# B&R Automation Studio project CarWash
Automation Studio 

## Configuration Config1

### Task classes (Cpu.sw)
```
Cyclic#1 (cycle 10000 us, tolerance 10000 us):
  Auxillary <- Source.Auxillary.Auxillary.prg
  MainCtrl <- Source.MainCtrl.MainCtrl.prg
  HPolish <- Source.Hpol.HPolish.prg
  EntryCtrl <- Source.Entrance.EntryCtrl.prg
  ChemCtrl <- Source.Chemicals.ChemCtrl.prg
  HPWater <- Source.HPWater.HPWater.prg
  HBrushCtrl <- Source.HBrush.HBrushCtrl.prg
  VBrushCtrl <- Source.VBrush.VBrushCtrl.prg
  UBCtrl <- Source.OptUnderBody.UBCtrl.prg
  VPolishCtr <- Source.OptVpolish.VPolishCtrl.prg
  WaxCtrl <- Source.OptWax.WaxCtrl.prg
  DryHCtrl <- Source.Drying.DryHCtrl.prg
  CarExit <- Source.CarExit.CarExit.prg
  AlarmCtrl <- Source.Infrastructure.AlarmCtrl.AlarmCtrl.prg
  DataCtrl <- Source.Infrastructure.DataCtrl.DataCtrl.prg
  RecipeCtrl <- Source.Infrastructure.RecipeCtrl.RecipeCtrl.prg
  VisuCtrl <- Source.VisuCtrl.VisuCtrl.prg
Cyclic#4 (cycle 100000 us, tolerance 100000 us):
  ComTCP_P <- Libraries.ComTCP.ComTCP_P.prg
Libraries: ComTCP_L, AsTCP, operator, runtime, astime, standard, ArEventLog, AsBrStr
```

### Hardware
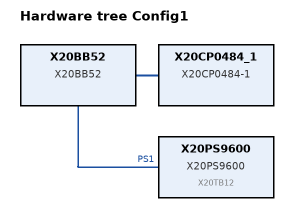
```
X20BB52 : X20BB52 v1.2.0.0
X20CP0484_1 : X20CP0484-1 v1.4.0.0  [SL -> X20BB52.SL1]
  Connector IF2:
    ActivateDevice = 1
  ConfigurationID = CarWashSimu_Config1
  Simulation = 1
  TimerDeviceType = SWIOTIMER
  Cyclic1Duration = 10000
  Cyclic1Tolerance = 10000
  Cyclic2Duration = 20000
  Cyclic2Tolerance = 20000
  Cyclic3Duration = 50000
  Cyclic3Tolerance = 50000
  Cyclic4Duration = 100000
  Cyclic4Tolerance = 100000
  Cyclic5Duration = 200000
  Cyclic5Tolerance = 200000
  Cyclic6Duration = 500000
  Cyclic6Tolerance = 500000
  Cyclic7Duration = 1000000
  Cyclic7Tolerance = 1000000
  Cyclic8Duration = 10000
  Cyclic8Tolerance = 30000000
  FileDevice1
  FileDeviceName1 = USER
  FileDevicePath1 = USER_PATH
X20PS9600 : X20PS9600 v1.6.0.0  [PS -> X20BB52.PS1; SS1 -> X20TB12.SS]
X20TB12 : X20TB12 v1.0.0.0
```

### PvMap.vvm - X20CP0484_1/PvMap.vvm
```iecst
VAR_CONFIG
<<<<<<< HEAD
	::CarExit:iExit.IO.doOrangeLight AT %Q.::ComTCP_SimOutputs.doExitOrangeLight; (*Insert your comment here...*)
	::CarExit:iExit.IO.doRedLight AT %Q.::ComTCP_SimOutputs.doExitRedLight; (*Insert your comment here...*)
	::ComTCP_SimOutputs.doExitGreenLight AT %Q.::ComTCP_SimOutputs.doExitGreenLight; (*Insert your comment here...*)
	::ComTCP_SimOutputs.doExitLiftDoorRelay AT %Q.::CarExit:iExit.IO.doRelayLiftDoor; (*Insert your comment here...*)
	::CarExit:iExit.IO.doRelayLowerdDoor AT %Q.::ComTCP_SimOutputs.doExitLowerDoorRelay; (*Insert your comment here...*)
	::MainCtrl:ScalDirt.y AT %Q.::ChemCtrl:iChem.IO.aoChemChemValve; (*Insert your comment here...*)
=======
	::VBrushCtrl:iVBrush.Par.LeftVel AT %Q.::ComTCP_SimOutputs.aoVBrushLVel; (*Insert your comment here...*)
	::VBrushCtrl:iVBrush.Par.RightVel AT %Q.::ComTCP_SimOutputs.aoVBrushRVel; (*Insert your comment here...*)
	::Auxillary:iAuxillary.doRelayConv AT %Q.::ComTCP_SimOutputs.doConvRelay; (*Insert your comment here...*)
	::ChemCtrl:iChem.IO.doChemWaterValve AT %Q.::ComTCP_SimOutputs.doChemWaterValve; (*Insert your comment here...*)
>>>>>>> edcf355ccd2dc5a058ed4214cc82538d90d7c920
	::ComTCP_SimInputs.aiEntranceSoilLevel AT %Q.::EntryCtrl:iEntry.IO.diSensSoilLvl; (*Insert your comment here...*)
	::ComTCP_SimInputs.aiVBrushLForceF AT %Q.::VBrushCtrl:iVBrush.IO.aiVBLForceF; (*Insert your comment here...*)
	::ComTCP_SimInputs.aiVBrushLForceS AT %Q.::VBrushCtrl:iVBrush.IO.aiVBLForceS; (*Insert your comment here...*)
	::ComTCP_SimInputs.aiVBrushRForceF AT %Q.::VBrushCtrl:iVBrush.IO.aiVBRForceF; (*Insert your comment here...*)
	::ComTCP_SimInputs.aiVBrushRForceS AT %Q.::VBrushCtrl:iVBrush.IO.aiVBRForceS; (*Insert your comment here...*)
	::ComTCP_SimInputs.diEmergencyStop AT %Q.::MainCtrl:gMain.Cmd.EStop; (*Insert your comment here...*)
	::ComTCP_SimInputs.diEntranceSensor AT %Q.::EntryCtrl:iEntry.IO.diSensEntry; (*Insert your comment here...*)
	::ComTCP_SimInputs.diHBrushSensor1 AT %Q.::HBrushCtrl:iHBrush.IO.diSensHB1; (*Insert your comment here...*)
	::ComTCP_SimInputs.diHBrushSensor2 AT %Q.::HBrushCtrl:iHBrush.IO.diSensHB2; (*Insert your comment here...*)
	::ComTCP_SimInputs.diHBrushSensor3 AT %Q.::HBrushCtrl:iHBrush.IO.diSensHB3; (*Insert your comment here...*)
	::ComTCP_SimInputs.diHBrushSensor4 AT %Q.::HBrushCtrl:iHBrush.IO.diSensHB4; (*Insert your comment here...*)
	::ComTCP_SimInputs.diHighPressSensor1 AT %Q.::HPWater:iHighPress.IO.diSensHP1; (*Insert your comment here...*)
	::ComTCP_SimInputs.diHighPressSensor2 AT %Q.::HPWater:iHighPress.IO.diSensHP2; (*Insert your comment here...*)
	::ComTCP_SimInputs.diHighPressSensor3 AT %Q.::HPWater:iHighPress.IO.diSensHP3; (*Insert your comment here...*)
	::ComTCP_SimInputs.diHighPressSensor4 AT %Q.::HPWater:iHighPress.IO.diSensHP4; (*Insert your comment here...*)
	::ComTCP_SimInputs.diHPolishSensor1 AT %Q.::HPolish:iHPolish.IO.diSensHPolish1; (*Insert your comment here...*)
	::ComTCP_SimInputs.diHPolishSensor2 AT %Q.::HPolish:iHPolish.IO.diSensHPolish2; (*Insert your comment here...*)
	::ComTCP_SimInputs.diHPolishSensor3 AT %Q.::HPolish:iHPolish.IO.diSensHPolish3; (*Insert your comment here...*)
	::ComTCP_SimInputs.diHPolishSensor4 AT %Q.::HPolish:iHPolish.IO.diSensHPolish4; (*Insert your comment here...*)
	::HBrushCtrl:iHBrush.IO.doRelayHBBrush AT %Q.::ComTCP_SimOutputs.doHBrushBrushRelay; (*Insert your comment here...*)
	::HBrushCtrl:iHBrush.IO.doRelayHBLift AT %Q.::ComTCP_SimOutputs.doHBrushLiftRelay; (*Insert your comment here...*)
	::HBrushCtrl:iHBrush.IO.doRelayHBLower AT %Q.::ComTCP_SimOutputs.doHBrushLowerRelay; (*Insert your comment here...*)
	::HBrushCtrl:iHBrush.IO.doValveHB AT %Q.::ComTCP_SimOutputs.doHBrushValve; (*Insert your comment here...*)
	::HPolish:iHPolish.IO.doRelayBrush AT %Q.::ComTCP_SimOutputs.doHPolishBrushRelay; (*Insert your comment here...*)
	::HPolish:iHPolish.IO.doRelayLift AT %Q.::ComTCP_SimOutputs.doHPolishLiftRelay; (*Insert your comment here...*)
	::HPolish:iHPolish.IO.doRelayLower AT %Q.::ComTCP_SimOutputs.doHPolishLowerRelay; (*Insert your comment here...*)
	::HPWater:iHighPress.IO.doRelayHPLift AT %Q.::ComTCP_SimOutputs.doHighPressLiftRelay; (*Insert your comment here...*)
	::HPWater:iHighPress.IO.doRelayHPLow AT %Q.::ComTCP_SimOutputs.doHighPressLowerRelay; (*Insert your comment here...*)
	::HPWater:iHighPress.IO.doRelayHPPump AT %Q.::ComTCP_SimOutputs.doHighPressPumpRelay; (*Insert your comment here...*)
	::HPWater:iHighPress.IO.doValveHP AT %Q.::ComTCP_SimOutputs.doHighPressValve; (*Insert your comment here...*)
	::MainCtrl:ScalDirt.y AT %Q.::ChemCtrl:iChem.IO.aoChemChemValve; (*Insert your comment here...*)
	::UBCtrl:iUBody.IO.doRelayPump AT %Q.::ComTCP_SimOutputs.doUnderbodyPumpRelay; (*Insert your comment here...*)
	::UBCtrl:iUBody.IO.doValveUB AT %Q.::ComTCP_SimOutputs.doUnderbodyValve; (*Insert your comment here...*)
	::VBrushCtrl:iVBrush.IO.doRelayVBLClose AT %Q.::ComTCP_SimOutputs.doVBrushRelayLClose; (*Insert your comment here...*)
	::VBrushCtrl:iVBrush.IO.doRelayVBLOpen AT %Q.::ComTCP_SimOutputs.doVBrushRelayLOpen; (*Insert your comment here...*)
	::VBrushCtrl:iVBrush.IO.doRelayVBRClose AT %Q.::ComTCP_SimOutputs.doVBrushRelayRClose; (*Insert your comment here...*)
	::VBrushCtrl:iVBrush.IO.doRelayVBROpen AT %Q.::ComTCP_SimOutputs.doVBrushRelayROpen; (*Insert your comment here...*)
<<<<<<< HEAD
	::VBrushCtrl:iVBrush.IO.doRelayVBLOpen AT %Q.::ComTCP_SimOutputs.doVBrushRelayLOpen; (*Insert your comment here...*)
	::ComTCP_SimInputs.aiVBrushLForceF AT %Q.::VBrushCtrl:iVBrush.IO.aiVBLForceF; (*Insert your comment here...*)
	::ComTCP_SimInputs.aiVBrushRForceF AT %Q.::VBrushCtrl:iVBrush.IO.aiVBRForceF; (*Insert your comment here...*)
	::ComTCP_SimInputs.aiVBrushLForceS AT %Q.::VBrushCtrl:iVBrush.IO.aiVBLForceS; (*Insert your comment here...*)
	::ComTCP_SimInputs.aiVBrushRForceS AT %Q.::VBrushCtrl:iVBrush.IO.aiVBRForceS; (*Insert your comment here...*)
	::ComTCP_SimInputs.diHDry1Sensor1 AT %Q.::DryHCtrl:iDry.IO.diSens1Dry1; (*Insert your comment here...*)
	::ComTCP_SimInputs.diHDry1Sensor2 AT %Q.::DryHCtrl:iDry.IO.diSens1Dry2; (*Insert your comment here...*)
	::ComTCP_SimInputs.diHDry1Sensor3 AT %Q.::DryHCtrl:iDry.IO.diSens1Dry3; (*Insert your comment here...*)
	::ComTCP_SimInputs.diHDry1Sensor4 AT %Q.::DryHCtrl:iDry.IO.diSens1Dry4; (*Insert your comment here...*)
	::ComTCP_SimInputs.diHDry2Sensor1 AT %Q.::DryHCtrl:iDry.IO.diSens2Dry1; (*Insert your comment here...*)
	::ComTCP_SimInputs.diHDry2Sensor2 AT %Q.::DryHCtrl:iDry.IO.diSens2Dry2; (*Insert your comment here...*)
	::ComTCP_SimInputs.diHDry2Sensor3 AT %Q.::DryHCtrl:iDry.IO.diSens2Dry3; (*Insert your comment here...*)
	::ComTCP_SimInputs.diHDry2Sensor4 AT %Q.::DryHCtrl:iDry.IO.diSens2Dry4; (*Insert your comment here...*)
	::DryHCtrl:iDry.IO.doRelayHD1Vent AT %Q.::ComTCP_SimOutputs.doHDry1VentRelay; (*Insert your comment here...*)
	::DryHCtrl:iDry.IO.doRelayHD1Heater AT %Q.::ComTCP_SimOutputs.doHDry1HeaterRelay; (*Insert your comment here...*)
	::DryHCtrl:iDry.IO.doRelayHD1Lower AT %Q.::ComTCP_SimOutputs.doHDry1LowerRelay; (*Insert your comment here...*)
	::DryHCtrl:iDry.IO.doRelayHD1Lift AT %Q.::ComTCP_SimOutputs.doHDry1LiftRelay; (*Insert your comment here...*)
	::DryHCtrl:iDry.IO.doRelayHD2Vent AT %Q.::ComTCP_SimOutputs.doHDry2VentRelay; (*Insert your comment here...*)
	::DryHCtrl:iDry.IO.doRelayHD2Heater AT %Q.::ComTCP_SimOutputs.doHDry2HeaterRelay; (*Insert your comment here...*)
	::DryHCtrl:iDry.IO.doRelayHD2Lower AT %Q.::ComTCP_SimOutputs.doHDry2LowerRelay; (*Insert your comment here...*)
	::DryHCtrl:iDry.IO.doRelayVDHeater AT %Q.::ComTCP_SimOutputs.doVDry1HeaterRelay; (*Insert your comment here...*)
	::DryHCtrl:iDry.IO.doRelayVDVent AT %Q.::ComTCP_SimOutputs.doVDry1VentRelay; (*Insert your comment here...*)
	::DryHCtrl:iDry.IO.doRelayHD2Lift AT %Q.::ComTCP_SimOutputs.doHDry2LiftRelay; (*Insert your comment here...*)
=======
	::WaxCtrl:iWax.IO.doValveWax AT %Q.::ComTCP_SimOutputs.doWaxValve; (*Insert your comment here...*)
	::WaxCtrl:iWax.IO.doRefillWax AT %Q.::ComTCP_SimOutputs.doWaxRefill; (*Insert your comment here...*)
	::WaxCtrl:iWax.IO.doRealyWaxPump AT %Q.::ComTCP_SimOutputs.doWaxPumpRelay; (*Insert your comment here...*)
>>>>>>> edcf355ccd2dc5a058ed4214cc82538d90d7c920
END_VAR
```

## Logical view

Binary libraries used (declarations not repeated): operator, runtime, astime, AsIecCon, AsTCP, standard, ArEventLog, AsBrStr, LoopConR, sys_lib, brsystem

### Package Logical/Libraries - Global libraries

### Library Logical/Libraries/ComTCP/ComTCP_L (ANSIC)
Depends on: AsTCP, operator, runtime, astime, standard, ArEventLog, AsBrStr

### Program Logical/Source/MainCtrl/MainCtrl

#### Types.typ
```iecst
TYPE
	sMainStep_enum1 :
		(
		enWAIT,
		enSTART,
		enENTRY,
		enCHEMICAL
		);
	MainCmd_typ : 	STRUCT
		Start : BOOL;
		Stop : BOOL;
		EStop : BOOL;
	END_STRUCT;
	MainOption_typ : 	STRUCT
		EntryState : BOOL;
		ChemicalState : BOOL;
		HighPress : BOOL;
		HBrush : BOOL;
		Polish : BOOL;
	END_STRUCT;
	MainCtrl_typ : 	STRUCT
		Cmd : MainCmd_typ;
		Option : MainOption_typ;
	END_STRUCT;
END_TYPE
```

#### Variables.var
```iecst
VAR
	ScalDirt : LCRScal;
	Status2 : UINT; (*status*)
	pEntryCtrl : REFERENCE TO EntryCtrl_typ; (*pointer*)
	SizeChem : UDINT; (*size of foil*)
	ChemAddress : UDINT; (*Address of foil*)
	pChemCtrl : REFERENCE TO ChemCtrl_typ; (*pointer*)
	SizeEntry : UDINT; (*size of foil*)
	EntryAddress : UDINT; (*Address of foil*)
	New_Variable : USINT;
	Car : INT;
	Status3 : UINT; (*status*)
	Status1 : UINT; (*status*)
	i : INT;
	SizeAux : UDINT;
	AuxAddress : UDINT;
	pAuxCtrl : REFERENCE TO Auxillary_typ;
	txt : WSTRING[80];
	txt1 : WSTRING[80];
	iFb_Timer : ARRAY[0..2] OF TON := [3((PT:=T#147720ms))];
	Status4 : UINT;
	HPAddress : UDINT;
	SizeHP : UDINT;
	pHPCtrl : REFERENCE TO HPWaterCtrl_typ;
	gMain : MainCtrl_typ;
	Status5 : UINT;
	HBAddress : UDINT;
	SizeHBrush : UDINT;
	pHBrushCtrl : REFERENCE TO HBrushCtrl_typ;
	Status6 : UINT;
	HPolishAddress : UDINT;
	SizeHPolish : UDINT;
	pHPolish : REFERENCE TO PolishCtrl_typ;
END_VAR
```

#### Main.st
```iecst
PROGRAM _INIT

	//accessing structre and data from tasks
	Status1 := PV_xgetadr(ADR('EntryCtrl:iEntry'),ADR(EntryAddress),ADR(SizeEntry));
	Status2 := PV_xgetadr(ADR('ChemCtrl:iChem'),ADR(ChemAddress),ADR(SizeChem));
	Status3 := PV_xgetadr(ADR('Auxillary:iAuxillary'),ADR(AuxAddress),ADR(SizeAux));
	Status4	:= PV_xgetadr(ADR('HPWater:iHighPress'), ADR(HPAddress), ADR(SizeHP));
	Status5	:= PV_xgetadr(ADR('HBrushCtrl:iHBrush'), ADR(HBAddress), ADR(SizeHBrush));
	Status6	:= PV_xgetadr(ADR('HPolish:iHPolish'), ADR(HPolishAddress), ADR(SizeHPolish));

END_PROGRAM

PROGRAM _CYCLIC
	//accessing data from the address
	pEntryCtrl ACCESS EntryAddress;
	pChemCtrl ACCESS ChemAddress;
	pAuxCtrl ACCESS AuxAddress;
	pHPCtrl ACCESS HPAddress;
	pHBrushCtrl ACCESS HBAddress;
	pHPolish ACCESS HPolishAddress;

	ScalDirt(x:=pEntryCtrl.IO.diSensSoilLvl ,y1:=5,x2:=10,y2:=0);

	IF gMain.Cmd.Start = TRUE THEN
		pAuxCtrl.doRelayConv	:= TRUE;
		gMain.Cmd.Start			:= FALSE;
		gMain.Option.EntryState	:= TRUE;
		FOR i:=0 TO 3 DO
			IF gCar[i]=FALSE THEN
				gCar[i]:=TRUE;
				EXIT;
			END_IF;
		END_FOR;
	END_IF;

	IF (gMain.Option.EntryState = TRUE) THEN

		pEntryCtrl.Cmd.Start:=TRUE;
		txt:="entry";

		IF pEntryCtrl.IO.diSensEntry=TRUE THEN
			iFb_Timer[0].IN:=TRUE;
		END_IF;

	END_IF;

	IF (iFb_Timer[0].ET >T#5400ms) AND (gMain.Option.ChemicalState = TRUE) THEN
		gMain.Option.EntryState			:= FALSE;
		txt:="chem";
		pChemCtrl.IO.doChemWaterValve	:= TRUE;
	END_IF;

	IF iFb_Timer[0].ET > (T#5400ms + T#11000ms) THEN
		pChemCtrl.IO.doChemWaterValve	:= FALSE;
		gMain.Option.ChemicalState		:= FALSE;
	END_IF;

	IF (iFb_Timer[0].ET > T#18290ms) AND (gMain.Option.HighPress = TRUE) THEN
		txt:="HighPressure Water";
		pHPCtrl.Cmd.Start		:= TRUE;
	END_IF;

	IF (iFb_Timer[0].ET > T#30650ms) AND (gMain.Option.HBrush = TRUE) THEN
		txt	:= "Horizontal Brush";
		pHBrushCtrl.Cmd.Start	:= TRUE;
		gMain.Option.HighPress	:= FALSE;
	END_IF;

	IF (iFb_Timer[0].ET > T#30650ms) AND (gMain.Option.HBrush = TRUE) THEN
		txt	:= "Horizontal Brush";
		pHBrushCtrl.Cmd.Start	:= TRUE;
		gMain.Option.HighPress	:= FALSE;
	END_IF;

	IF (iFb_Timer[0].ET > T#72000ms) AND (gMain.Option.Polish = TRUE) THEN
		txt	:= "Polishing";
		pHPolish.Cmd.Start	:= TRUE;
		gMain.Option.HBrush	:= FALSE;
	END_IF;

	IF gMain.Cmd.EStop = TRUE THEN
		iFb_Timer[0]();
	END_IF;

END_PROGRAM

PROGRAM _EXIT
	(* Insert code here *)

END_PROGRAM
```

### EntryCtrl.typ
```iecst
TYPE
	EntryCmd_typ : 	STRUCT
		Start : BOOL;
		EStop : BOOL;
		Stop : BOOL;
	END_STRUCT;
	EntryCtrl_typ : 	STRUCT
		Cmd : EntryCmd_typ;
		IO : EntryIOs_typ;
		Par : EntryParam_typ;
		Status : EntryStatus_typ;
	END_STRUCT;
	EntryIOs_typ : 	STRUCT
		diSensEntry : BOOL;
		diSensSoilLvl : REAL;
	END_STRUCT;
	EntryParam_typ : 	STRUCT
		CarLength : REAL;
	END_STRUCT;
	EntryStatus_typ : 	STRUCT
		Running : BOOL;
		Error : BOOL;
		CarGone : BOOL;
		CarIN : BOOL;
	END_STRUCT;
END_TYPE
```

### Program Logical/Source/Entrance/EntryCtrl

#### Variables.var
```iecst
VAR
	iEntry : EntryCtrl_typ;
	value : sStep;
	iEntryState : sStep;
END_VAR
```

#### Main.st
```iecst
PROGRAM _INIT
	(* Insert code here *)

END_PROGRAM

PROGRAM _CYCLIC
	(* Insert code here *)
	iEntry;

	CASE iEntryState OF

		enWAIT:

			IF iEntry.Cmd.Start=TRUE THEN
				iEntryState:=enSTART;
			END_IF;

		enSTART:
			IF iEntry.IO.diSensEntry=TRUE THEN
				iEntryState:=enCARIN;
			END_IF;
		enCARIN:
			iEntry.Status.CarGone:=FALSE;
			iEntry.Status.CarIN:=TRUE;

			IF iEntry.IO.diSensEntry=FALSE THEN
				iEntry.Status.CarIN:=FALSE;
				iEntry.Status.CarGone:=TRUE;
				iEntryState:=enWAIT;
			END_IF;

		enERROR:

	END_CASE;
END_PROGRAM

PROGRAM _EXIT
	(* Insert code here *)

END_PROGRAM
```

### ChemCtrl.typ
```iecst
TYPE
	ChemCmd_typ : 	STRUCT
		Start : BOOL;
		EStop : BOOL;
		Stop : BOOL;
	END_STRUCT;
	ChemCtrl_typ : 	STRUCT
		Cmd : ChemCmd_typ;
		IO : ChemIOs_typ;
		Par : ChemParam_typ;
		Status : ChemStatus_typ;
	END_STRUCT;
	ChemIOs_typ : 	STRUCT
		aoChemChemValve : REAL;
		doChemWaterValve : BOOL;
		doChemRefill : BOOL;
	END_STRUCT;
	ChemParam_typ : 	STRUCT
		ChemLevel : REAL;
	END_STRUCT;
	ChemStatus_typ : 	STRUCT
		Running : BOOL;
		Error : BOOL;
		ChemHigh : BOOL;
		ChemLow : BOOL;
	END_STRUCT;
END_TYPE
```

### Program Logical/Source/Chemicals/ChemCtrl

#### Types.typ
```iecst
TYPE
	sStep_enum :
		(
		enWAIT,
		enSTART,
		enSPRAYON,
		enSPRAYOFF,
		enERROR
		);
END_TYPE
```

#### Main.st
```iecst
PROGRAM _INIT
	(* Insert code here *)

END_PROGRAM

PROGRAM _CYCLIC
	(* Insert code here *)
	iChem.Par.ChemLevel:=ScalDirt.y;

	CASE sChemState OF

		enWAIT:
			iChem.Status.Running:=FALSE;
			sChemState:=enSTART;

		enSTART:

		enSPRAYON:

		enSPRAYOFF:

	END_CASE;
END_PROGRAM

PROGRAM _EXIT
	(* Insert code here *)

END_PROGRAM
```

### HPWater.typ
```iecst
TYPE
	HPWaterCmd_typ : 	STRUCT
		Start : BOOL;
		EStop : BOOL;
		Stop : BOOL;
	END_STRUCT;
	HPWaterCtrl_typ : 	STRUCT
		Cmd : HPWaterCmd_typ;
		IO : HPWaterIOs_typ;
		Par : HPWaterParam_typ;
		Status : HPWaterStatus_typ;
	END_STRUCT;
	HPWaterIOs_typ : 	STRUCT
		diSensHP1 : BOOL;
		diSensHP2 : BOOL;
		diSensHP3 : BOOL;
		diSensHP4 : BOOL;
		doValveHP : BOOL;
		doRelayHPPump : BOOL;
		doRelayHPLow : BOOL;
		doRelayHPLift : BOOL;
	END_STRUCT;
	HPWaterParam_typ : 	STRUCT
		New_Member : USINT;
	END_STRUCT;
	HPWaterStatus_typ : 	STRUCT
		Running : BOOL;
		Error : BOOL;
		ValveOpen : USINT;
		New_Member6 : USINT;
		New_Member5 : USINT;
		New_Member4 : USINT;
		New_Member3 : USINT;
		New_Member2 : USINT;
		New_Member1 : USINT;
		New_Member : USINT;
	END_STRUCT;
END_TYPE
```

### Program Logical/Source/HPWater/HPWater

#### Types.typ
```iecst
TYPE
	HighPressureState_enum :
		(
		enWAIT,
		enSTART,
		enLIFTDOWN,
		enLIFTSTABLE,
		enLIFTUP,
		enERROR
		);
END_TYPE
```

#### Variables.var
```iecst
VAR
	sHighPressState : HighPressureState_enum;
END_VAR
```

#### Main.st
```iecst
PROGRAM _INIT
	(* Insert code here *)

END_PROGRAM

PROGRAM _CYCLIC
	(* Insert code here *)

	CASE sHighPressState OF
		enWAIT:
		IF

	END_CASE;

END_PROGRAM

PROGRAM _EXIT
	(* Insert code here *)

END_PROGRAM
```

### HBrushCtrl.typ
```iecst
TYPE
	HBrushCmd_typ : 	STRUCT
		Start : BOOL;
		EStop : BOOL;
		Stop : BOOL;
	END_STRUCT;
	HBrushCtrl_typ : 	STRUCT
		Cmd : HBrushCmd_typ;
		IO : HBrushIOs_typ;
		Par : HBrushParam_typ;
		Status : HBrushStatus_typ;
	END_STRUCT;
	HBrushIOs_typ : 	STRUCT
	END_STRUCT;
	HBrushParam_typ : 	STRUCT
	END_STRUCT;
	HBrushStatus_typ : 	STRUCT
		Running : BOOL;
		Error : BOOL;
	END_STRUCT;
END_TYPE
```

### Program Logical/Source/HBrush/HBrushCtrl

#### Variables.var
```iecst
VAR
	iHBrush : HBrushCtrl_typ;
	sHBrushState : HorizonBrushState_enum;
END_VAR
```

#### Main.st
```iecst
PROGRAM _INIT
	(* Insert code here *)

END_PROGRAM

PROGRAM _CYCLIC
	(* Insert code here *)
	CASE sHBrushState OF
		enWAIT:
			IF iHBrush.Cmd.Start = TRUE THEN
				sHBrushState				:= enSTART;
				iHBrush.IO.doValveHB		:= TRUE;
			END_IF;
		enSTART:
			IF (iHBrush.IO.diSensHB1 = FALSE) AND (iHBrush.IO.diSensHB2 = FALSE) AND (iHBrush.IO.diSensHB3 = FALSE) AND (iHBrush.IO.diSensHB4 = FALSE) THEN
				iHBrush.IO.doRelayHBLower	:= TRUE;
				iHBrush.IO.doRelayHBLift	:= FALSE;
			END_IF;
			IF (iHBrush.IO.diSensHB1 = TRUE) AND (iHBrush.IO.diSensHB2 = FALSE) AND (iHBrush.IO.diSensHB3 = FALSE) AND (iHBrush.IO.diSensHB4 = FALSE) THEN
				iHBrush.IO.doRelayHBLower	:= FALSE;
				iHBrush.IO.doRelayHBLift	:= FALSE;
				iHBrush.IO.doRelayHBBrush	:= TRUE;
				sHBrushState				:= enOPERATION;
			END_IF;
		enOPERATION:
			IF (iHBrush.IO.diSensHB1 = TRUE) AND (iHBrush.IO.diSensHB2 = FALSE) AND (iHBrush.IO.diSensHB3 = FALSE) AND (iHBrush.IO.diSensHB4 = FALSE) THEN
				iHBrush.IO.doRelayHBLower	:= FALSE;
				iHBrush.IO.doRelayHBLift	:= FALSE;
			END_IF;
			IF (iHBrush.IO.diSensHB1 = TRUE) AND (iHBrush.IO.diSensHB2 = TRUE) AND (iHBrush.IO.diSensHB3 = TRUE) AND (iHBrush.IO.diSensHB4 = FALSE) THEN
				iHBrush.IO.doRelayHBLower	:= FALSE;
				iHBrush.IO.doRelayHBLift	:= TRUE;
			END_IF;
			IF (iHBrush.IO.diSensHB1 = TRUE) AND (iHBrush.IO.diSensHB2 = TRUE) AND (iHBrush.IO.diSensHB3 = FALSE) AND (iHBrush.IO.diSensHB4 = FALSE) THEN
				iHBrush.IO.doRelayHBLower	:= FALSE;
				iHBrush.IO.doRelayHBLift	:= TRUE;
			END_IF;
			IF (iHBrush.IO.diSensHB1 = FALSE) AND (iHBrush.IO.diSensHB2 = FALSE) AND (iHBrush.IO.diSensHB3 = TRUE) AND (iHBrush.IO.diSensHB4 = FALSE) THEN
				iHBrush.IO.doRelayHBLower	:= TRUE;
				iHBrush.IO.doRelayHBLift	:= FALSE;
			END_IF;
			IF (iHBrush.IO.diSensHB1 = FALSE) AND (iHBrush.IO.diSensHB2 = FALSE) AND (iHBrush.IO.diSensHB3 = TRUE) AND (iHBrush.IO.diSensHB4 = TRUE) THEN
				iHBrush.IO.doRelayHBLower	:= FALSE;
				iHBrush.IO.doRelayHBLift	:= FALSE;
			END_IF;
			IF (iHBrush.IO.diSensHB1 = FALSE) AND (iHBrush.IO.diSensHB2 = FALSE) AND (iHBrush.IO.diSensHB3 = FALSE) AND (iHBrush.IO.diSensHB4 = FALSE) THEN
				iHBrush.IO.doRelayHBLower	:= FALSE;
				iHBrush.IO.doRelayHBLift	:= FALSE;
				iHBrush.IO.doRelayHBBrush	:= FALSE;
				iHBrush.IO.doValveHB		:= FALSE;
				iHBrush.Cmd.Start		:= FALSE;
				sHBrushState				:= enWAIT;
			END_IF;

	END_CASE;

END_PROGRAM

PROGRAM _EXIT
	(* Insert code here *)

END_PROGRAM
```

### VBrushCtrl.typ
```iecst
TYPE
	VBrushCmd_typ : 	STRUCT
		Start : BOOL;
		EStop : BOOL;
		Stop : BOOL;
	END_STRUCT;
	VBrushCtrl_typ : 	STRUCT
		Cmd : VBrushCmd_typ;
		IO : VBrushIOs_typ;
		Par : VBrushParam_typ;
		Status : VBrushStatus_typ;
	END_STRUCT;
	VBrushIOs_typ : 	STRUCT
		doRelayVBLClose : BOOL;
		doRelayVBROpen : BOOL;
		doRelayVBLOpen : BOOL;
		doRelayVBRClose : BOOL;
		aiVBRForceS : REAL;
		aiVBRForceF : REAL;
		aiVBLForceS : REAL;
		aiVBLForceF : REAL;
		aoVBRRVelocity : REAL;
		aoVBRLVelocity : REAL;
	END_STRUCT;
	VBrushParam_typ : 	STRUCT
		Velocity : USINT;
	END_STRUCT;
	VBrushStatus_typ : 	STRUCT
		Running : BOOL;
		Error : BOOL;
		ForceIN : BOOL;
		Rotating : USINT;
	END_STRUCT;
END_TYPE
```

### Program Logical/Source/VBrush/VBrushCtrl

#### Types.typ
```iecst
TYPE
	sStep_enum :
		(
		enWAIT,
		enOPERATION,
		enERROR
		);
END_TYPE
```

#### Main.st
```iecst
PROGRAM _INIT
	(* Insert code here *)

END_PROGRAM

PROGRAM _CYCLIC
	(* Insert code here *)

END_PROGRAM

PROGRAM _EXIT
	(* Insert code here *)

END_PROGRAM
```

### UBCtrl.typ
```iecst
TYPE
	UBCmd_typ : 	STRUCT
		Start : BOOL;
		EStop : BOOL;
		Stop : BOOL;
	END_STRUCT;
	UBCtrl_typ : 	STRUCT
		Cmd : UBCmd_typ;
		IO : UBIOs_typ;
		Par : UBParam_typ;
		Status : UBStatus_typ;
	END_STRUCT;
	UBIOs_typ : 	STRUCT
		doValveUB : BOOL;
		doRelayPump : BOOL;
	END_STRUCT;
	UBParam_typ : 	STRUCT
	END_STRUCT;
	UBStatus_typ : 	STRUCT
		Running : BOOL;
		Error : BOOL;
		PumpOpen : BOOL;
		ValveOpen : BOOL;
	END_STRUCT;
END_TYPE
```

### WaxCtrl.typ
```iecst
TYPE
	WaxCmd_typ : 	STRUCT
		Start : BOOL;
		EStop : BOOL;
		Stop : BOOL;
	END_STRUCT;
	WaxCtrl_typ : 	STRUCT
		Cmd : WaxCmd_typ;
		IO : WaxIOs_typ;
		Par : WaxParam_typ;
		Status : WaxStatus_typ;
	END_STRUCT;
	WaxIOs_typ : 	STRUCT
		doValveWax : USINT;
		doRealyWaxPump : USINT;
		doRefillWax : USINT;
	END_STRUCT;
	WaxParam_typ : 	STRUCT
	END_STRUCT;
	WaxStatus_typ : 	STRUCT
		Running : BOOL;
		Error : BOOL;
		PumpOn : BOOL;
		ValveOpen : BOOL;
	END_STRUCT;
END_TYPE
```

### DryCtrl.typ
```iecst
TYPE
	DryCmd_typ : 	STRUCT
		Start : BOOL;
		EStop : BOOL;
		Stop : BOOL;
	END_STRUCT;
	DryCtrl_typ : 	STRUCT
		Cmd : DryCmd_typ;
		IO : DryIOs_typ;
		Par : DryParam_typ;
		Status : DryStatus_typ;
	END_STRUCT;
	DryIOs_typ : 	STRUCT
		diSensDry1 : BOOL;
		diSensDry2 : BOOL;
		diSensDry3 : BOOL;
		diSensDry4 : BOOL;
		diSens2Dry2 : BOOL;
		diSens2Dry3 : BOOL;
		diSens2Dry4 : BOOL;
		diSens2Dry1 : BOOL;
		doRelayHD1Lower : BOOL;
		doRelayHD1LVent1 : BOOL;
		doRelayHD1Heater1 : BOOL;
		doRelayVDLVent : BOOL;
		doRelayVDHeater : BOOL;
		doRelayHD1Lift : BOOL;
		doRelayHD2Lower : BOOL;
		doRelayHD2LVent : BOOL;
		doRelayHD2Heater : BOOL;
		doRelayHD2Lift : BOOL;
	END_STRUCT;
	DryParam_typ : 	STRUCT
	END_STRUCT;
	DryStatus_typ : 	STRUCT
		Running : BOOL;
		Error : BOOL;
	END_STRUCT;
END_TYPE
```

### CarExit.typ
```iecst
TYPE
	CarExitCmd_typ : 	STRUCT
		Start : BOOL;
		EStop : BOOL;
		Stop : BOOL;
	END_STRUCT;
	CarExitCtrl_typ : 	STRUCT
		Cmd : CarExitCmd_typ;
		IO : CarExitIOs_typ;
		Par : CarExitParam_typ;
		Status : CarExitStatus_typ;
	END_STRUCT;
	CarExitIOs_typ : 	STRUCT
		doGreenLight : BOOL;
		doRelayLowerdDoor : BOOL;
		doRelayLiftDoor : BOOL;
		doRedLight : BOOL;
		doOrangeLight : BOOL;
	END_STRUCT;
	CarExitParam_typ : 	STRUCT
	END_STRUCT;
	CarExitStatus_typ : 	STRUCT
		Running : BOOL;
		Error : BOOL;
		LiftingDoor : BOOL;
		LowringDoor : BOOL;
	END_STRUCT;
END_TYPE
```

- Visualisation Logical/Source/VisuCtrl (not shown)

### HPolishCtrl.typ
```iecst
TYPE
	PolishCmd_typ : 	STRUCT
		Start : BOOL;
		EStop : BOOL;
		Stop : BOOL;
	END_STRUCT;
	PolishCtrl_typ : 	STRUCT
		Cmd : PolishCmd_typ;
		IO : PolishIOs_typ;
		Par : PolishParam_typ;
		Status : PolishStatus_typ;
	END_STRUCT;
	PolishIOs_typ : 	STRUCT
		doRelayLower : USINT;
		doRelayBrush : USINT;
		doRelayLift : USINT;
	END_STRUCT;
	PolishParam_typ : 	STRUCT
	END_STRUCT;
	PolishStatus_typ : 	STRUCT
		Running : BOOL;
		Error : BOOL;
	END_STRUCT;
END_TYPE
```

### Program Logical/Source/Optpolish/HPolishCtrl (IEC)

#### Main.st
```iecst
PROGRAM _INIT
	(* Insert code here *)

END_PROGRAM

PROGRAM _CYCLIC
iHPolish;
END_PROGRAM

PROGRAM _EXIT
	(* Insert code here *)

END_PROGRAM
```

### HPolishCtrl.typ
```iecst
TYPE
	PolishCmd_typ : 	STRUCT
		Start : BOOL;
		EStop : BOOL;
		Stop : BOOL;
	END_STRUCT;
	PolishCtrl_typ : 	STRUCT
		Cmd : PolishCmd_typ;
		IO : PolishIOs_typ;
		Par : PolishParam_typ;
		Status : PolishStatus_typ;
	END_STRUCT;
	PolishIOs_typ : 	STRUCT
		doRelayLower : USINT;
		doRelayBrush : USINT;
		doRelayLift : USINT;
	END_STRUCT;
	PolishParam_typ : 	STRUCT
		New_Member : USINT;
	END_STRUCT;
	PolishStatus_typ : 	STRUCT
		Running : BOOL;
		Error : BOOL;
	END_STRUCT;
END_TYPE
```

### PolishCtrl.typ - not listed in the package file held
```iecst
TYPE
	PolishCmd_typ : 	STRUCT
		Start : BOOL;
		EStop : BOOL;
		Stop : BOOL;
	END_STRUCT;
	PolishCtrl_typ : 	STRUCT
		Cmd : PolishCmd_typ;
		IO : PolishIOs_typ;
		Par : PolishParam_typ;
		Status : PolishStatus_typ;
	END_STRUCT;
	PolishIOs_typ : 	STRUCT
	END_STRUCT;
	PolishParam_typ : 	STRUCT
	END_STRUCT;
	PolishStatus_typ : 	STRUCT
		Running : BOOL;
		Error : BOOL;
	END_STRUCT;
END_TYPE
```

### Program Logical/Dist

#### Main.st
```iecst
PROGRAM _INIT
	(* Insert code here *)

END_PROGRAM

PROGRAM _CYCLIC
	a	:= a + 0.44;
END_PROGRAM

PROGRAM _EXIT
	(* Insert code here *)

END_PROGRAM
```

### Program Logical/Main

#### Variables.var
```iecst
VAR
	a : BOOL;
	b : BOOL;
END_VAR
```

#### Main.st
```iecst
PROGRAM _INIT
	(* Insert code here *)

END_PROGRAM

PROGRAM _CYCLIC
	(* Insert code here *)
	IF a = TRUE THEN
		b := TRUE;
	END_IF;

END_PROGRAM

PROGRAM _EXIT
	(* Insert code here *)

END_PROGRAM
```

Listed in the project but not available here: Logical/Global.typ, Logical/Global.var, Logical/Libraries/ComTCP/ComTCP_L/MNG_InternalTyp.hpp, Logical/Libraries/ComTCP/ComTCP_L/MNG_ComHdlr.hpp, Logical/Libraries/ComTCP/ComTCP_L/MNG_ComHdlr.cpp, Logical/Libraries/ComTCP/ComTCP_L/MNG_Global.hpp, Logical/Libraries/ComTCP/ComTCP_L/MNG_CpyOutToMsg.cpp, Logical/Libraries/ComTCP/ComTCP_L/MNG_CpyMsgToInp.cpp, Logical/Libraries/ComTCP/ComTCP_P, Logical/Libraries/ComTCP/MNG_Package.typ, Logical/Libraries/ComTCP/MNG_Package.var, Logical/MNG_Global.typ, Logical/Documentation, Logical/Source/OptVpolish, Logical/Source/Drying/DryHCtrl, Logical/Source/Drying/DryVCtrl, Logical/Source/Infrastructure, Logical/Source/Hpol, Logical/Source/Auxillary
